(*
SPDX-FileCopyrightText: © 2026 Oleksandr Tiutyk <trofimich@gmail.com>
SPDX-License-Identifier: MIT
License: https://opensource.org/license/mit
*)

INTERFACE IEvent EXTENDS IObject

{attribute 'monitoring' := 'call'}
PROPERTY Handled : BOOL
GET
END_GET
END_PROPERTY

METHOD SetHandled
END_METHOD

{attribute 'monitoring' := 'call'}
PROPERTY SourceObject : IObject
GET
END_GET
END_PROPERTY

END_INTERFACE

(* stored: Version 1.1.0.1
   Itf IEvent: Id {4290fe22-bbfe-42ca-acfa-29f4b1a003dc}
   Property Handled: Id {887baed9-f1ee-4209-9b76-3b844d59fcde}
   Get Get: Id {4825f4b2-b919-4f9b-9c79-4e4388a5282d}
   Method SetHandled: Id {bf90052d-8d4e-4a65-a834-1f380b97a326}
   Property SourceObject: Id {f823d641-dad4-46f7-8bef-0714c45a8a9b}
   Get Get: Id {c4b87340-f526-4515-8c1c-13ce336c21d0} *)
